GLOBALCONSTANTS STATES (* Global constants *)
  (* Standard: 61499-1; Description: Copyright (c) 2025 HR Agrartechnik GmbH This program and the accompanying materials are made available under the terms of the Eclipse Public License 2.0 which is available at https://www.eclipse.org/legal/epl-2.0/ SPDX-License-Identifier: EPL-2.0 *)
  (* Version 1.0, 2025-05-23, Franz Höpfinger, HR Agrartechnik GmbH *)
  PACKAGE Verteiler::LinksRechts;
  VAR_GLOBAL CONSTANT
    Rechtslauf : STRING := STRING#'Rechtslauf';
    Linkslauf : STRING := STRING#'Linkslauf';
    Linkslauf_Pause : STRING := STRING#'Linkslauf_Pause';
    Rechtslauf_Pause : STRING := STRING#'Rechtslauf_Pause';
  END_VAR
END_GLOBALCONSTANTS
